// TIA Portal V20 export
FUNCTION_BLOCK "FB_BwLoader"   // FB88, SCL
{ S7_Optimized_Access := 'TRUE' }
// stored: MemoryReserve 100, SetENOAutomatically false
   VAR
      sBwCommunication : "FB_BwCommunication";
      sTONBW_CtrlInProgress { S7_SetPoint := 'True'} : TP_TIME;
   END_VAR
BEGIN
   REGION Description header 
       //==================================================================================
       // POSALUX Swiss SA / (C) Copyright 2024
       //----------------------------------------------------------------------------------
       // Title: FB_BwLoader
       // Comment/Function: 
       //
       // Author: Fabien WALDT
       // Engineering: TIA Portal v20
       //----------------------------------------------------------------------------------
       // Change log table:
       // Version  | Date     | Expert in charge | Changes applied
       // ---------|----------|------------------|------------------------------------
       // 00.00.01 | 20260127 | WFA              | First released version
       // ==================================================================================
   END_REGION

   REGION Inputs Update
       "DB_BwLoaderExchange".Inputs.LifeFlag := "AI_LifeFlag";
       IF NOT #sBwCommunication.oLifeFlagError THEN
           "DB_BwLoaderExchange".Inputs.JobDone := "DI_JobDone";
           "DB_BwLoaderExchange".Inputs.LockShuttle := "DI_LockShuttle";
           "DB_BwLoaderExchange".Inputs.DataSend := "AI_DataSend";
           "DB_BwLoaderExchange".Inputs.DataReceive := "AI_DataReceive";
           "DB_BwLoaderExchange".Inputs.NoEmergencyStopAtBwLoader := "DI_NoEmergencyStopAtBwLoader";
           "DB_BwLoaderExchange".Inputs.SafetyDoorsClosedAtBwLoader := "DI_SafetyDoorsClosedAtBwLoader";
           "DB_BwLoaderExchange".Inputs.BwInErrorState := "AI_BwInErrorState";
           "DB_BwLoaderExchange".Inputs.UndrilledPartControl := "DI_UndrilledPartControl";
           "DB_BwLoaderExchange".Inputs.DrilledPartControl := "DI_DrilledPartControl";
           "DB_BwLoaderExchange".Inputs.BackwallControl := "DI_BackwallControl";
           "DB_BwLoaderExchange".Inputs.BwLoaderInSafePos := "DI_BwLoaderInSafePos";
       ELSE
           "DB_BwLoaderExchange".Inputs.JobDone := FALSE;
           "DB_BwLoaderExchange".Inputs.LockShuttle := FALSE;
           "DB_BwLoaderExchange".Inputs.DataSend := 0;
           "DB_BwLoaderExchange".Inputs.DataReceive := 0;
           "DB_BwLoaderExchange".Inputs.NoEmergencyStopAtBwLoader := FALSE;
           "DB_BwLoaderExchange".Inputs.SafetyDoorsClosedAtBwLoader := FALSE;
           "DB_BwLoaderExchange".Inputs.BwInErrorState := 0;
           "DB_BwLoaderExchange".Inputs.UndrilledPartControl := FALSE;
           "DB_BwLoaderExchange".Inputs.DrilledPartControl := FALSE;
           "DB_BwLoaderExchange".Inputs.BackwallControl := FALSE;
           "DB_BwLoaderExchange".Inputs.BwLoaderInSafePos := FALSE;
       END_IF;
   END_REGION

   REGION
       #sBwCommunication(iShuttle1Load := "DB_LoaderShuttle1".sBwLoadUnload.oBwLoadReq,
                         iShuttle1Unload := "DB_LoaderShuttle1".sBwLoadUnload.oBwUnloadReq,
                         iShuttle2Load := "DB_LoaderShuttle2".sBwLoadUnload.oBwLoadReq,
                         iShuttle2Unload := "DB_LoaderShuttle2".sBwLoadUnload.oBwUnloadReq,
                         iFromBwLoaderLifeFlag := "DB_BwLoaderExchange".Inputs.LifeFlag,
                         iFromBwLoaderJobDone := "DB_BwLoaderExchange".Inputs.JobDone,
                         iFromBwLoaderLockShuttle := "DB_BwLoaderExchange".Inputs.LockShuttle,
                         iFromBwLoaderDatasR := "DB_BwLoaderExchange".Inputs.DataReceive,
                         iFromBwLoaderDatasS:="DB_BwLoaderExchange".Inputs.DataSend,
                         iBwInErrorState:="DB_BwLoaderExchange".Inputs.BwInErrorState,
                         oLoadJobDone => #sBwCommunication.oLoadJobDone,
                         oUnloadJobDone => #sBwCommunication.oUnloadJobDone,
                         oLifeFlagError => #sBwCommunication.oLifeFlagError,
                         ioToBwLoaderLifeFlag := "DB_BwLoaderExchange".Outputs.LifeFlag,
                         ioToBwLoaderLoaderRequest := "DB_BwLoaderExchange".Outputs.LoaderRequest,
                         ioToBwLoaderLockShuttle := "DB_BwLoaderExchange".Outputs.LockShuttle,
                         ioToBwLoaderDatas := "DB_BwLoaderExchange".Outputs.DataSend);
      END_REGION

      REGION Alarmes
          // Défaut communication Chargeur de Backwall
          IF #sBwCommunication.oLifeFlagError THEN
              "LBP_AlarmMsgs".UserA[03].A70UUxx[28] := TRUE;
          END_IF;

          // Défaut général Chargeur de Backwall
          "LBP_AlarmMsgs".UserA[03].A70UUxx[29] := #sBwCommunication.iBwInErrorState <> 0;
      END_REGION

      REGION Outputs management
          "DB_BwLoaderExchange".Outputs.NoEmergencyStopAtFemto := NOT "DB_DataFromSafety".EmergencyStop;
          "DB_BwLoaderExchange".Outputs.SafetyDoorsClosedAtFemto := "DB_DataFromSafety".DoorsClosed;

          IF "DB_Alarms".sAlarmsLevel6 THEN
              "DB_BwLoaderExchange".Outputs.FemtoInErrorState := 6;
          ELSIF "DB_Alarms".sAlarmsLevel5 THEN
              "DB_BwLoaderExchange".Outputs.FemtoInErrorState := 5;
          ELSIF "DB_Alarms".sAlarmsLevel4 THEN
              "DB_BwLoaderExchange".Outputs.FemtoInErrorState := 4;
          ELSIF "DB_Alarms".sAlarmsLevel3 THEN
              "DB_BwLoaderExchange".Outputs.FemtoInErrorState := 3;
          ELSIF "DB_Alarms".sAlarmsLevel2 THEN
              "DB_BwLoaderExchange".Outputs.FemtoInErrorState := 2;
          ELSIF "DB_Alarms".sAlarmsLevel1 THEN
              "DB_BwLoaderExchange".Outputs.FemtoInErrorState := 1;
          ELSE
              "DB_BwLoaderExchange".Outputs.FemtoInErrorState := 1;
          END_IF;

          "DB_BwLoaderExchange".Outputs.AutoMode := "LBP_ModeGroup".E_AUTO;
          "DB_BwLoaderExchange".Outputs.JogMode := "LBP_ModeGroup".E_JOG;
          "DB_BwLoaderExchange".Outputs.GotoSafePos := "LBP_Chan1".A_Ref;
          "DB_BwLoaderExchange".Outputs.Emptying := "DB_WorkingModes".sEmptying;
      END_REGION

      REGION BW Control IN in progress
          "DB_BwLoaderExchange".Outputs.BW_CtrlInProgress :=
          ("DB_AxisPosition".sAxis05_U1."$AA_IM" = "DB_AxisPosMachinePLC".Axis_U1.BwControl AND "DB_LoaderShuttle1".sBwControlIn.sCurrent_Step_NB <> 0)
          OR ("DB_AxisPosition".sAxis06_U2."$AA_IM" = "DB_AxisPosMachinePLC".Axis_U2.BwControl AND "DB_LoaderShuttle2".sBwControlIn.sCurrent_Step_NB <> 0);
      END_REGION

      REGION  Outputs Update
          "AQ_LifeFlag" := "DB_BwLoaderExchange".Outputs.LifeFlag;
          "DQ_LoaderRequest":= "DB_BwLoaderExchange".Outputs.LoaderRequest;
          "DQ_LockShuttle" := "DB_BwLoaderExchange".Outputs.LockShuttle;
          "AQ_DataSend" := "DB_BwLoaderExchange".Outputs.DataSend;
          "AQ_DataReceive":= "DB_BwLoaderExchange".Outputs.DataReceive;
          "DQ_NoEmergencyStopAtFemto" := "DB_BwLoaderExchange".Outputs.NoEmergencyStopAtFemto;
          "DQ_SafetyDoorsClosedAtFemto" := "DB_BwLoaderExchange".Outputs.SafetyDoorsClosedAtFemto;
          "AQ_FemtoInErrorState" := "DB_BwLoaderExchange".Outputs.FemtoInErrorState;
          "DQ_AutoMode" :="DB_BwLoaderExchange".Outputs.AutoMode;
          "DQ_JogMode" := "DB_BwLoaderExchange".Outputs.JogMode;
          "DQ_GotoSafePos":= "DB_BwLoaderExchange".Outputs.GotoSafePos;
          "DQ_Emptying" := "DB_BwLoaderExchange".Outputs.Emptying;
          "DQ_BW_CtrlInProgress" := "DB_BwLoaderExchange".Outputs.BW_CtrlInProgress;
      END_REGION

      REGION Reset à supprimer
          IF "DB_McpKeyboardSignals".sAlarmReset.sKeySWStatus THEN
              "AQ_Reset" := 1;
          ELSIF "MCP1_In".reset THEN
              "AQ_Reset" := 2;
          ELSE
              "AQ_Reset" := 0;
          END_IF;
      END_REGION
END_FUNCTION_BLOCK
